KUKA KRL program: HP010.src, HP010.dat

--- HP010.src ---
&ACCESS RVP
&REL 2
&COMMENT ACCELO BOLHA
&PARAM TEMPLATE = C:\KRC\roboter\template\vg_hp
&PARAM EDITMASK = HP*
DEF HP010( )
;FOLD INI
  ;FOLD BASISTECH INI
    GLOBAL INTERRUPT DECL 3 WHEN $STOPMESS==TRUE DO IR_STOPM ( )
    INTERRUPT ON 3
    BAS (#INITMOV,0 )
  ;ENDFOLD (BASISTECH INI)
  ;FOLD GRIPPERTECH INI
    USER_GRP(0,DUMMY,DUMMY,GDEFAULT)
  ;ENDFOLD (GRIPPERTECH INI)

  ;FOLD USER INI
    ;Make your modifications here
     ;FOLD COLLISION_V_3.01 INI ;%{E}
        IF (COLLISION_DATA[1].I_NR>0) THEN
          GLOBAL INTERRUPT DECL 21 WHEN $IN[COLLISION_DATA[1].I_NR]==FALSE DO COLLSTOP (1,0 )
        ENDIF
        IF (COLLISION_DATA[2].I_NR>0) THEN
          GLOBAL INTERRUPT DECL 22 WHEN $IN[COLLISION_DATA[2].I_NR]==FALSE DO COLLSTOP (2,0 )
        ENDIF
        IF (COLLISION_DATA[3].I_NR>0) THEN
          GLOBAL INTERRUPT DECL 23 WHEN $IN[COLLISION_DATA[3].I_NR]==FALSE DO COLLSTOP (3,0 )
        ENDIF
        IF (COLLISION_DATA[4].I_NR>0) THEN
          GLOBAL INTERRUPT DECL 24 WHEN $IN[COLLISION_DATA[4].I_NR]==FALSE DO COLLSTOP (4,0 )
        ENDIF
     ;ENDFOLD (Collision)
  ;ENDFOLD (USER INI)
;ENDFOLD (INI)

; Caracterização dos meios de produção:
; Changes: Accelo Bolha
; Versão Atual: 03/11/2017
; Name: P13.050-R4

$TIMER[3]=0
$TIMER_STOP[3]=FALSE

chk_w8_wechs_ok ( )           ; CHECK FERRAMENTA: TOOL CHANGE

MBINI ( )                     ; RESET DE BITS

;FOLD PTP HOME  Vel= 100 % DEFAULT;%{PE}%MKUKATPBASIS,%CMOVE,%VPTP,%P 1:PTP, 2:HOME, 3:, 5:100, 7:DEFAULT
$BWDSTART = FALSE
$H_POS=XHOME
PDAT_ACT=PDEFAULT
BAS (#PTP_DAT )
FDAT_ACT=FHOME
BAS (#FRAMES )
BAS (#VEL_PTP,100 )
PTP  XHOME
;ENDFOLD

WKZ4_AN ( )                   ; PEGA GRIPPER ACCELO

HO_ST621_R4_2 ( )             ; PEGA FRONTAL ACCELO

AB_ST600_R4_2 ( )             ; DEPOSITA FRONTAL NA GEOB

WKZ1_AN ( )                   ; PEGA PINÇA C1

start_weld_GEO ( )            ; BIT DE SOLDA GEOMETRIA

ps_ltc_geo_c1 ( )             ; SOLDA GEOMETRIA C1

WKZ1_AB ( )                   ; DEPOSITA PINÇA C1

WKZ2_AN ( )                   ; PEGA PINÇA C2

ps_ltc_geo_c2_Bolha ( )       ; SOLDA GEOMETRIA C2

end_weld_GEO ( )              ; BIT FIM DE SOLDA GEOMETRIA

start_weld_RESPOT ( )         ; BIT INICIO DE SOLDA RESPOT

ps_ltc_res_c2 ( )             ; SOLDA RESPOT C2

WKZ2_AB ( )                   ; DEPOSITA PINÇA C2

WKZ4_OFF_ST600 ( )            ; PEGA GRIPPER NA GEO

end_weld_RESPOT ( )           ; BIT FIM DE SOLDA RESPOT

MBINI_2 ( )                   ; RESET DE BITS FINAIS

WKZ4_AB ( )                   ; DEPOSITA GRIPPER ACCELO

MBINI ( )                     ; RESET DE BITS INICIAIS

;FOLD PTP HOME  Vel= 100 % DEFAULT;%{PE}%MKUKATPBASIS,%CMOVE,%VPTP,%P 1:PTP, 2:HOME, 3:, 5:100, 7:DEFAULT
$BWDSTART = FALSE
$H_POS=XHOME
PDAT_ACT=PDEFAULT
BAS (#PTP_DAT )
FDAT_ACT=FHOME
BAS (#FRAMES )
BAS (#VEL_PTP,100 )
PTP  XHOME
;ENDFOLD  ; PONTO INTERMEDIÁRIO

$TIMER_STOP[3]=TRUE

END

--- HP010.dat ---
&ACCESS RVP
&REL 2
&COMMENT ACCELO BOLHA
&PARAM TEMPLATE = C:\KRC\roboter\template\vg_hp
&PARAM EDITMASK = HP*
DEFDAT HP010
;FOLD EXTERNAL DECLARATIONS;%{PE}%MKUKATPBASIS,%CEXT,%VCOMMON,%P
;FOLD BASISTECH EXT;%{PE}%MKUKATPBASIS,%CEXT,%VEXT,%P
EXT  BAS (BAS_COMMAND  :IN,REAL  :IN )
DECL INT SUCCESS
;ENDFOLD (BASISTECH EXT)
;FOLD GRIPPERTECH EXT
EXT  H50 (INT  :IN,INT  :IN,INT  :IN,GRP_TYP  :IN )
;ENDFOLD (GRIPPERTECH EXT)
;FOLD SPOTTECH EXT
EXT  USERSPOT (S_COMMAND  :IN,SPOT_TYPE  :IN )
;ENDFOLD (SPOTTECH EXT)
;FOLD USER EXT;%{E}%MKUKATPUSER,%CEXT,%VEXT,%P
;Make here your modifications

;FOLD COLLISION
EXT  COLLSTOP (INT  :IN,INT  :IN )
;ENDFOLD  (Collision)
;ENDFOLD (USER EXT)
;ENDFOLD (EXTERNAL DECLERATIONS)
DECL FDAT FHOME={TOOL_NO 0,BASE_NO 0,IPO_FRAME #BASE}
DECL BASIS_SUGG_T LAST_BASIS={POINT1[] "P1                      ",POINT2[] "P1                      ",CP_PARAMS[] "CPDAT0                  ",PTP_PARAMS[] "PDAT1                   ",CONT[] "C_DIS                   ",CP_VEL[] "2.0                     ",PTP_VEL[] "100                     ",SYNC_PARAMS[] "SYNCDAT                 ",SPL_NAME[] "S0                      "}
ENDDAT
